{attribute 'no_explicit_call' := 'no direct call necessary'}
PROGRAM PRG_TaskLog
VAR
	aTaskLogger			: ARRAY[1..SIZEOF(TwinCAT_SystemInfoVarList._TaskInfo)/SIZEOF(PlcTaskSystemInfo)] OF FB_Log4TcTask;
	aTaskRtcTime		: ARRAY[1..SIZEOF(TwinCAT_SystemInfoVarList._TaskInfo)/SIZEOF(PlcTaskSystemInfo)] OF FB_RTC_Sync;
END_VAR

(*
:Description: Sends collected log message of a single task to the service. 

This method must be called in each task which uses logging. It should be
called once a cycle.

**Example**

.. code:: 

    PRG_TaskLog.Call();
	
*)
METHOD PUBLIC Call
VAR
	nIdx	: DINT;
END_VAR
nIdx := Tc2_Utilities.GETCURTASKINDEXEX();
aTaskLogger[nIdx].Call();
aTaskRtcTime[nIdx].Call();
END_METHOD

(*
:Description: Initialise the task logger with custom parameter. 

This method must be called in each task which uses logging. As long as
the parameter do not change a single call is sufficient.

**Example**

.. code:: 

	IF _TaskInfo[GETCURTASKINDEXEX()].FirstCycle THEN
		// For Remote Log4TC Server change the AMS net ID and configure a route
	  PRG_TaskLog.Init('127.0.0.1.1.1');
	END_IF
    
*)
METHOD PUBLIC Init : BOOL
VAR_INPUT
	sAmsNetId	: Tc2_Utilities.T_AmsNetID;	(* The ams net id of the log service. Defaults to localhost (empty string). *)
END_VAR
aTaskLogger[Tc2_Utilities.GETCURTASKINDEXEX()].Init(sAmsNetId);
END_METHOD

PROPERTY INTERNAL RtcTime : LINT
GET
RtcTime := aTaskRtcTime[Tc2_Utilities.GETCURTASKINDEXEX()].RtcTime;
END_GET
END_PROPERTY

(*
:Description: Returns the ``I_ContextBuilder`` for task specific context
	properties. 

Task specific properties are added to each log message which is created
on the same task. 

For best performance properties should only be added or removed if the
values have changed.

**Example**

.. code:: 

	IF _TaskInfo[GETCURTASKINDEXEX()].FirstCycle THEN
		PRG_TaskLog.TaskContextBuilder.AddInt('machineNo', nMachineNumber);
	END_IF
    
*)
PROPERTY PUBLIC TaskContextBuilder : I_ContextBuilder
GET
TaskContextBuilder := aTaskLogger[GETCURTASKINDEXEX()].TaskContext;
END_GET
END_PROPERTY

PROPERTY INTERNAL TaskLogger : REFERENCE TO FB_Log4TcTask
GET
TaskLogger REF= aTaskLogger[GETCURTASKINDEXEX()];
END_GET
END_PROPERTY

END_PROGRAM

(* stored: Version 1.1.0.1, ProductVersion 3.1.4024.0
   POU PRG_TaskLog: Id {d9deec54-041b-4d4a-a876-7d0487674ab5}, SpecialFunc None
   Method Call: Id {7aeb9926-c091-4a02-a0d3-9930716cb4d1}
   Method Init: Id {a5681b61-7170-465c-b800-f922f70178d3}
   Property RtcTime: Id {3577743f-dcc4-455c-a535-d7ff2826b706}
   Get Get: Id {743e0e5a-c100-4c91-84fb-00ad8ebc0e39}
   Property TaskContextBuilder: Id {37ede606-5a7a-4581-9bfb-710648eb6050}
   Get Get: Id {0565efa6-0f30-4a5a-8d01-6c8dcd2d67fb}
   Property TaskLogger: Id {e5ae713c-f421-49cb-9871-258b1113ba41}
   Get Get: Id {2041d993-1b63-44b0-b94c-7510408823c4} *)
